FUNCTION_BLOCK EM_Seal_Shrink IMPLEMENTS  ITF_EM_Seal_Shrink
VAR_INPUT
END_VAR
VAR_OUTPUT
END_VAR
VAR
END_VAR

END_FUNCTION_BLOCK

(* stored: Version 1.1.0.1, ProductVersion 3.1.4024.12
   POU EM_Seal_Shrink: Id {5aae22ce-6da8-45b3-8569-19b73574cdf0}, SpecialFunc None *)
